PROGRAM SyncProgram
VAR
	fbAxisSync : ContinousSync;
	bStartButton : BOOL;
	bStopButton : BOOL;
END_VAR

fbAxisSync.bStart := bStartButton;
fbAxisSync.bStop := bStopButton;

fbAxisSync();

END_PROGRAM

(* stored: Version 1.1.0.1, ProductVersion 3.1.4024.12
   POU SyncProgram: Id {69812283-6bdf-46df-860b-8389d106e3be}, SpecialFunc None *)
